(* PLC project service_side, Dassault Systèmes ControlBuild 2024x *)
(* stored: creationDateTime 2023-10-03T11:13:50-01:00 *)

FUNCTION_BLOCK tni_train.service_side
  VAR_OUTPUT
    rightServiceSide : BOOL := false;
    leftServiceSide : BOOL := true;
  END_VAR
  VAR
    button : BOOL := false;
  END_VAR

INITIAL_STEP 10:
  10_INLINE1(N);
  COMPUTE_FUNCTION_BLOCKS(S);
END_STEP
ACTION 10_INLINE1:
  leftServiceSide;
END_ACTION
TRANSITION FROM 10 TO 11
  := button;
END_TRANSITION
STEP 11:
  11_INLINE2(N);
END_STEP
ACTION 11_INLINE2:
  rightServiceSide;
END_ACTION
TRANSITION FROM 11 TO 10
  := NOT button;
END_TRANSITION
ACTION COMPUTE_FUNCTION_BLOCKS:  (* blocks drawn on the SFC sheet *)
  G1:
END_ACTION
END_FUNCTION_BLOCK
